REGION Network 50: End if not ready to next step
   // no SCL statement known for JumpNot: written as a call
   JumpNot(in := #POWER_STATE >= 90, label := END);
END_REGION

REGION Network 51: OPERATION
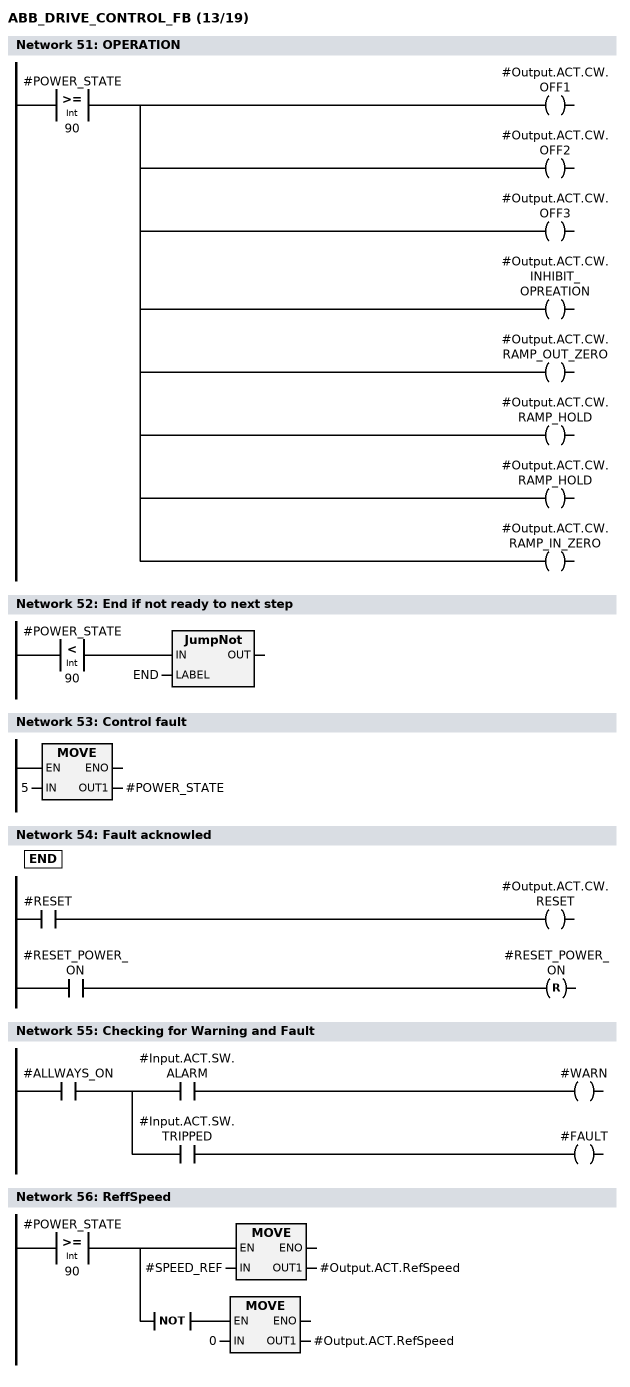
   RUNG wire#powerrail
      { S7_Templates := "SrcType := Int" } GE_Contact(in1 := #POWER_STATE, in2 := 90)
      wire#w1
      Coil( #Output.ACT.CW.OFF1 )
   END_RUNG
   RUNG wire#w1
      Coil( #Output.ACT.CW.OFF2 )
   END_RUNG
   RUNG wire#w1
      Coil( #Output.ACT.CW.OFF3 )
   END_RUNG
   RUNG wire#w1
      Coil( #Output.ACT.CW.INHIBIT_OPREATION )
   END_RUNG
   RUNG wire#w1
      Coil( #Output.ACT.CW.RAMP_OUT_ZERO )
   END_RUNG
   RUNG wire#w1
      Coil( #Output.ACT.CW.RAMP_HOLD )
   END_RUNG
   RUNG wire#w1
      Coil( #Output.ACT.CW.RAMP_HOLD )
   END_RUNG
   RUNG wire#w1
      Coil( #Output.ACT.CW.RAMP_IN_ZERO )
   END_RUNG
   // the same network as SCL:
   #Output.ACT.CW.OFF1 := #POWER_STATE >= 90;
   #Output.ACT.CW.OFF2 := #Output.ACT.CW.OFF1;
   #Output.ACT.CW.OFF3 := #Output.ACT.CW.OFF1;
   #Output.ACT.CW.INHIBIT_OPREATION := #Output.ACT.CW.OFF1;
   #Output.ACT.CW.RAMP_OUT_ZERO := #Output.ACT.CW.OFF1;
   #Output.ACT.CW.RAMP_HOLD := #Output.ACT.CW.OFF1;
   #Output.ACT.CW.RAMP_HOLD := #Output.ACT.CW.OFF1;
   #Output.ACT.CW.RAMP_IN_ZERO := #Output.ACT.CW.OFF1;
END_REGION

REGION Network 52: End if not ready to next step
   // no SCL statement known for JumpNot: written as a call
   JumpNot(in := #POWER_STATE < 90, label := END);
END_REGION

REGION Network 53: Control fault
   RUNG wire#powerrail
      { S7_GenerateENO := "TRUE" } Move(in := 5, out1 => #POWER_STATE)
   END_RUNG
   // the same network as SCL:
   #POWER_STATE := 5;
END_REGION

REGION Network 54: Fault acknowled
   Label( END )
   RUNG wire#powerrail
      Contact( #RESET )
      Coil( #Output.ACT.CW.RESET )
   END_RUNG
   RUNG wire#powerrail
      Contact( #RESET_POWER_ON )
      R_Coil( #RESET_POWER_ON )
   END_RUNG
   // the same network as SCL:
   END:
   #Output.ACT.CW.RESET := #RESET;
   IF #RESET_POWER_ON THEN #RESET_POWER_ON := FALSE; END_IF;
END_REGION

REGION Network 55: Checking for Warning and Fault
   RUNG wire#powerrail
      Contact( #ALLWAYS_ON )
      wire#w1
      Contact( #Input.ACT.SW.ALARM )
      Coil( #WARN )
   END_RUNG
   RUNG wire#w1
      Contact( #Input.ACT.SW.TRIPPED )
      Coil( #FAULT )
   END_RUNG
   // the same network as SCL:
   #WARN := #ALLWAYS_ON AND #Input.ACT.SW.ALARM;
   #FAULT := #ALLWAYS_ON AND #Input.ACT.SW.TRIPPED;
END_REGION

REGION Network 56: ReffSpeed
   RUNG wire#powerrail
      { S7_Templates := "SrcType := Int" } GE_Contact(in1 := #POWER_STATE, in2 := 90)
      wire#w1
      { S7_GenerateENO := "TRUE" } Move(in := #SPEED_REF, out1 => #Output.ACT.RefSpeed)
   END_RUNG
   RUNG wire#w1
      Not()
      { S7_GenerateENO := "TRUE" } Move(in := 0, out1 => #Output.ACT.RefSpeed)
   END_RUNG
   // the same network as SCL:
   #_w1 := #POWER_STATE >= 90;
   IF #_w1 THEN #Output.ACT.RefSpeed := #SPEED_REF; END_IF;
   IF NOT #_w1 THEN #Output.ACT.RefSpeed := 0; END_IF;
END_REGION

REGION Network 57: Write values PPO1 Fixed area
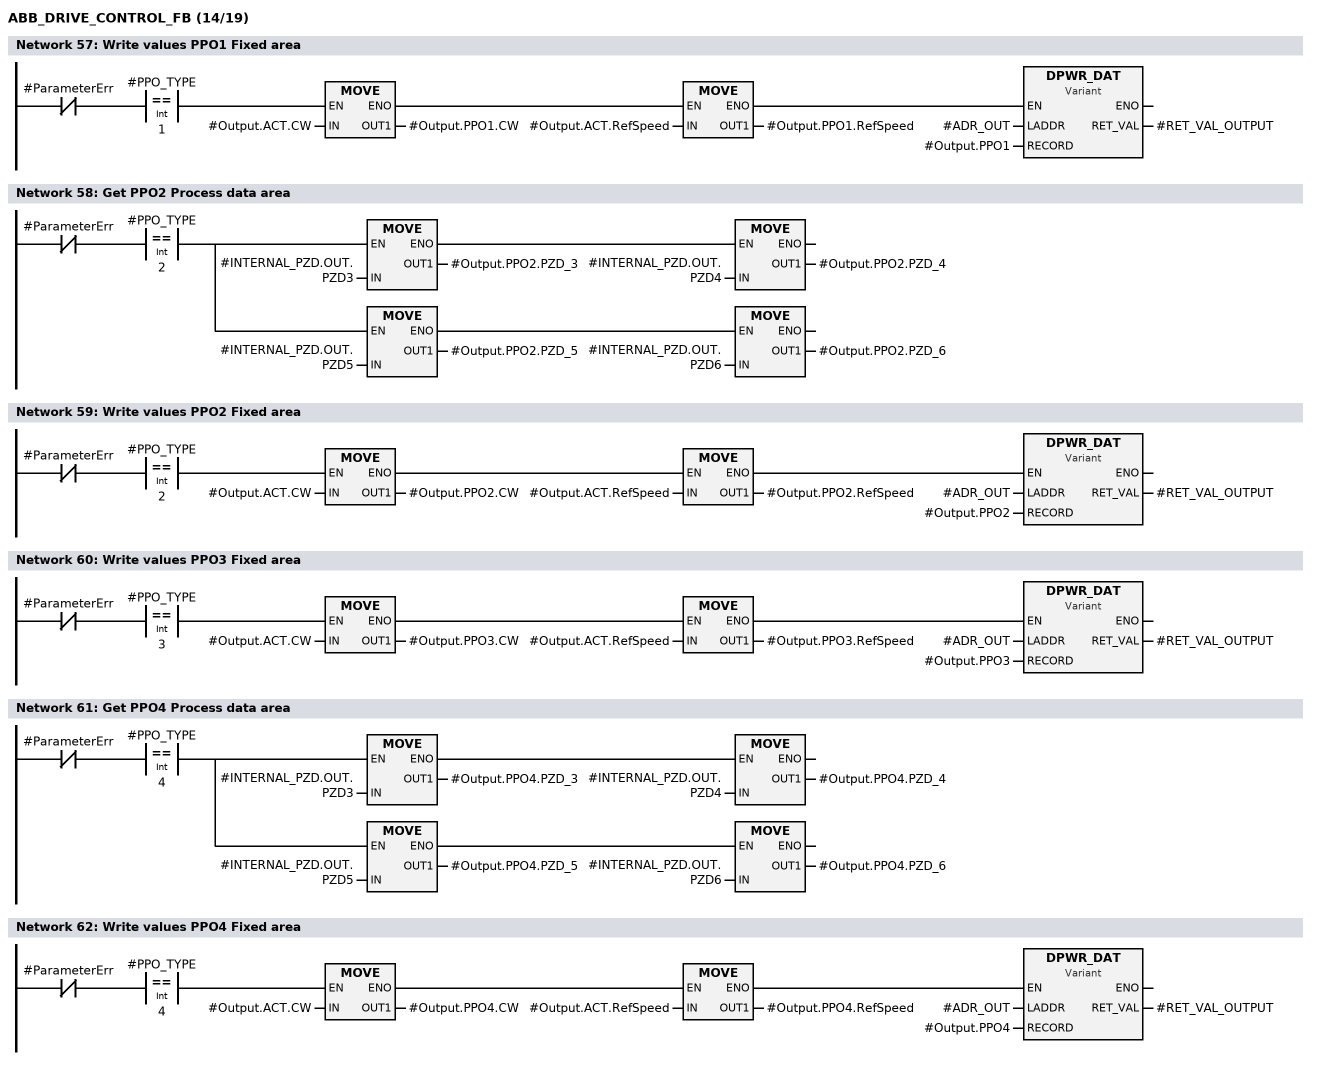
   RUNG wire#powerrail
      I_Contact( #ParameterErr )
      { S7_Templates := "SrcType := Int" } EQ_Contact(in1 := #PPO_TYPE, in2 := 1)
      { S7_GenerateENO := "TRUE" } Move(in := #Output.ACT.CW, out1 => #Output.PPO1.CW)
      { S7_GenerateENO := "TRUE" } Move(in := #Output.ACT.RefSpeed, out1 => #Output.PPO1.RefSpeed)
      { S7_Templates := "[ptr_type := Variant, laddr_type := HW_IO]" } DPWR_DAT(LADDR := #ADR_OUT, RECORD := #Output.PPO1, RET_VAL => #RET_VAL_OUTPUT)
   END_RUNG
   // the same network as SCL:
   // ENO of a box is taken as its EN; it also drops when the box reports an error
   IF NOT #ParameterErr AND (#PPO_TYPE = 1) THEN
       #Output.PPO1.CW := #Output.ACT.CW;
       #Output.PPO1.RefSpeed := #Output.ACT.RefSpeed;
       #RET_VAL_OUTPUT := DPWR_DAT(LADDR := #ADR_OUT, RECORD := #Output.PPO1);
   END_IF;
END_REGION

REGION Network 58: Get PPO2 Process data area
   RUNG wire#powerrail
      I_Contact( #ParameterErr )
      { S7_Templates := "SrcType := Int" } EQ_Contact(in1 := #PPO_TYPE, in2 := 2)
      wire#w1
      { S7_GenerateENO := "TRUE" } Move(in := #INTERNAL_PZD.OUT.PZD3, out1 => #Output.PPO2.PZD_3)
      { S7_GenerateENO := "TRUE" } Move(in := #INTERNAL_PZD.OUT.PZD4, out1 => #Output.PPO2.PZD_4)
   END_RUNG
   RUNG wire#w1
      { S7_GenerateENO := "TRUE" } Move(in := #INTERNAL_PZD.OUT.PZD5, out1 => #Output.PPO2.PZD_5)
      { S7_GenerateENO := "TRUE" } Move(in := #INTERNAL_PZD.OUT.PZD6, out1 => #Output.PPO2.PZD_6)
   END_RUNG
   // the same network as SCL:
   // ENO of a box is taken as its EN; it also drops when the box reports an error
   IF NOT #ParameterErr AND (#PPO_TYPE = 2) THEN
       #Output.PPO2.PZD_3 := #INTERNAL_PZD.OUT.PZD3;
       #Output.PPO2.PZD_4 := #INTERNAL_PZD.OUT.PZD4;
       #Output.PPO2.PZD_5 := #INTERNAL_PZD.OUT.PZD5;
       #Output.PPO2.PZD_6 := #INTERNAL_PZD.OUT.PZD6;
   END_IF;
END_REGION

REGION Network 59: Write values PPO2 Fixed area
   RUNG wire#powerrail
      I_Contact( #ParameterErr )
      { S7_Templates := "SrcType := Int" } EQ_Contact(in1 := #PPO_TYPE, in2 := 2)
      { S7_GenerateENO := "TRUE" } Move(in := #Output.ACT.CW, out1 => #Output.PPO2.CW)
      { S7_GenerateENO := "TRUE" } Move(in := #Output.ACT.RefSpeed, out1 => #Output.PPO2.RefSpeed)
      { S7_Templates := "[ptr_type := Variant, laddr_type := HW_IO]" } DPWR_DAT(LADDR := #ADR_OUT, RECORD := #Output.PPO2, RET_VAL => #RET_VAL_OUTPUT)
   END_RUNG
   // the same network as SCL:
   // ENO of a box is taken as its EN; it also drops when the box reports an error
   IF NOT #ParameterErr AND (#PPO_TYPE = 2) THEN
       #Output.PPO2.CW := #Output.ACT.CW;
       #Output.PPO2.RefSpeed := #Output.ACT.RefSpeed;
       #RET_VAL_OUTPUT := DPWR_DAT(LADDR := #ADR_OUT, RECORD := #Output.PPO2);
   END_IF;
END_REGION

REGION Network 60: Write values PPO3 Fixed area
   RUNG wire#powerrail
      I_Contact( #ParameterErr )
      { S7_Templates := "SrcType := Int" } EQ_Contact(in1 := #PPO_TYPE, in2 := 3)
      { S7_GenerateENO := "TRUE" } Move(in := #Output.ACT.CW, out1 => #Output.PPO3.CW)
      { S7_GenerateENO := "TRUE" } Move(in := #Output.ACT.RefSpeed, out1 => #Output.PPO3.RefSpeed)
      { S7_Templates := "[ptr_type := Variant, laddr_type := HW_IO]" } DPWR_DAT(LADDR := #ADR_OUT, RECORD := #Output.PPO3, RET_VAL => #RET_VAL_OUTPUT)
   END_RUNG
   // the same network as SCL:
   // ENO of a box is taken as its EN; it also drops when the box reports an error
   IF NOT #ParameterErr AND (#PPO_TYPE = 3) THEN
       #Output.PPO3.CW := #Output.ACT.CW;
       #Output.PPO3.RefSpeed := #Output.ACT.RefSpeed;
       #RET_VAL_OUTPUT := DPWR_DAT(LADDR := #ADR_OUT, RECORD := #Output.PPO3);
   END_IF;
END_REGION

REGION Network 61: Get PPO4 Process data area
   RUNG wire#powerrail
      I_Contact( #ParameterErr )
      { S7_Templates := "SrcType := Int" } EQ_Contact(in1 := #PPO_TYPE, in2 := 4)
      wire#w1
      { S7_GenerateENO := "TRUE" } Move(in := #INTERNAL_PZD.OUT.PZD3, out1 => #Output.PPO4.PZD_3)
      { S7_GenerateENO := "TRUE" } Move(in := #INTERNAL_PZD.OUT.PZD4, out1 => #Output.PPO4.PZD_4)
   END_RUNG
   RUNG wire#w1
      { S7_GenerateENO := "TRUE" } Move(in := #INTERNAL_PZD.OUT.PZD5, out1 => #Output.PPO4.PZD_5)
      { S7_GenerateENO := "TRUE" } Move(in := #INTERNAL_PZD.OUT.PZD6, out1 => #Output.PPO4.PZD_6)
   END_RUNG
   // the same network as SCL:
   // ENO of a box is taken as its EN; it also drops when the box reports an error
   IF NOT #ParameterErr AND (#PPO_TYPE = 4) THEN
       #Output.PPO4.PZD_3 := #INTERNAL_PZD.OUT.PZD3;
       #Output.PPO4.PZD_4 := #INTERNAL_PZD.OUT.PZD4;
       #Output.PPO4.PZD_5 := #INTERNAL_PZD.OUT.PZD5;
       #Output.PPO4.PZD_6 := #INTERNAL_PZD.OUT.PZD6;
   END_IF;
END_REGION

REGION Network 62: Write values PPO4 Fixed area
   RUNG wire#powerrail
      I_Contact( #ParameterErr )
      { S7_Templates := "SrcType := Int" } EQ_Contact(in1 := #PPO_TYPE, in2 := 4)
      { S7_GenerateENO := "TRUE" } Move(in := #Output.ACT.CW, out1 => #Output.PPO4.CW)
      { S7_GenerateENO := "TRUE" } Move(in := #Output.ACT.RefSpeed, out1 => #Output.PPO4.RefSpeed)
      { S7_Templates := "[ptr_type := Variant, laddr_type := HW_IO]" } DPWR_DAT(LADDR := #ADR_OUT, RECORD := #Output.PPO4, RET_VAL => #RET_VAL_OUTPUT)
   END_RUNG
   // the same network as SCL:
   // ENO of a box is taken as its EN; it also drops when the box reports an error
   IF NOT #ParameterErr AND (#PPO_TYPE = 4) THEN
       #Output.PPO4.CW := #Output.ACT.CW;
       #Output.PPO4.RefSpeed := #Output.ACT.RefSpeed;
       #RET_VAL_OUTPUT := DPWR_DAT(LADDR := #ADR_OUT, RECORD := #Output.PPO4);
   END_IF;
END_REGION

REGION Network 63: Get PPO5 Process data area
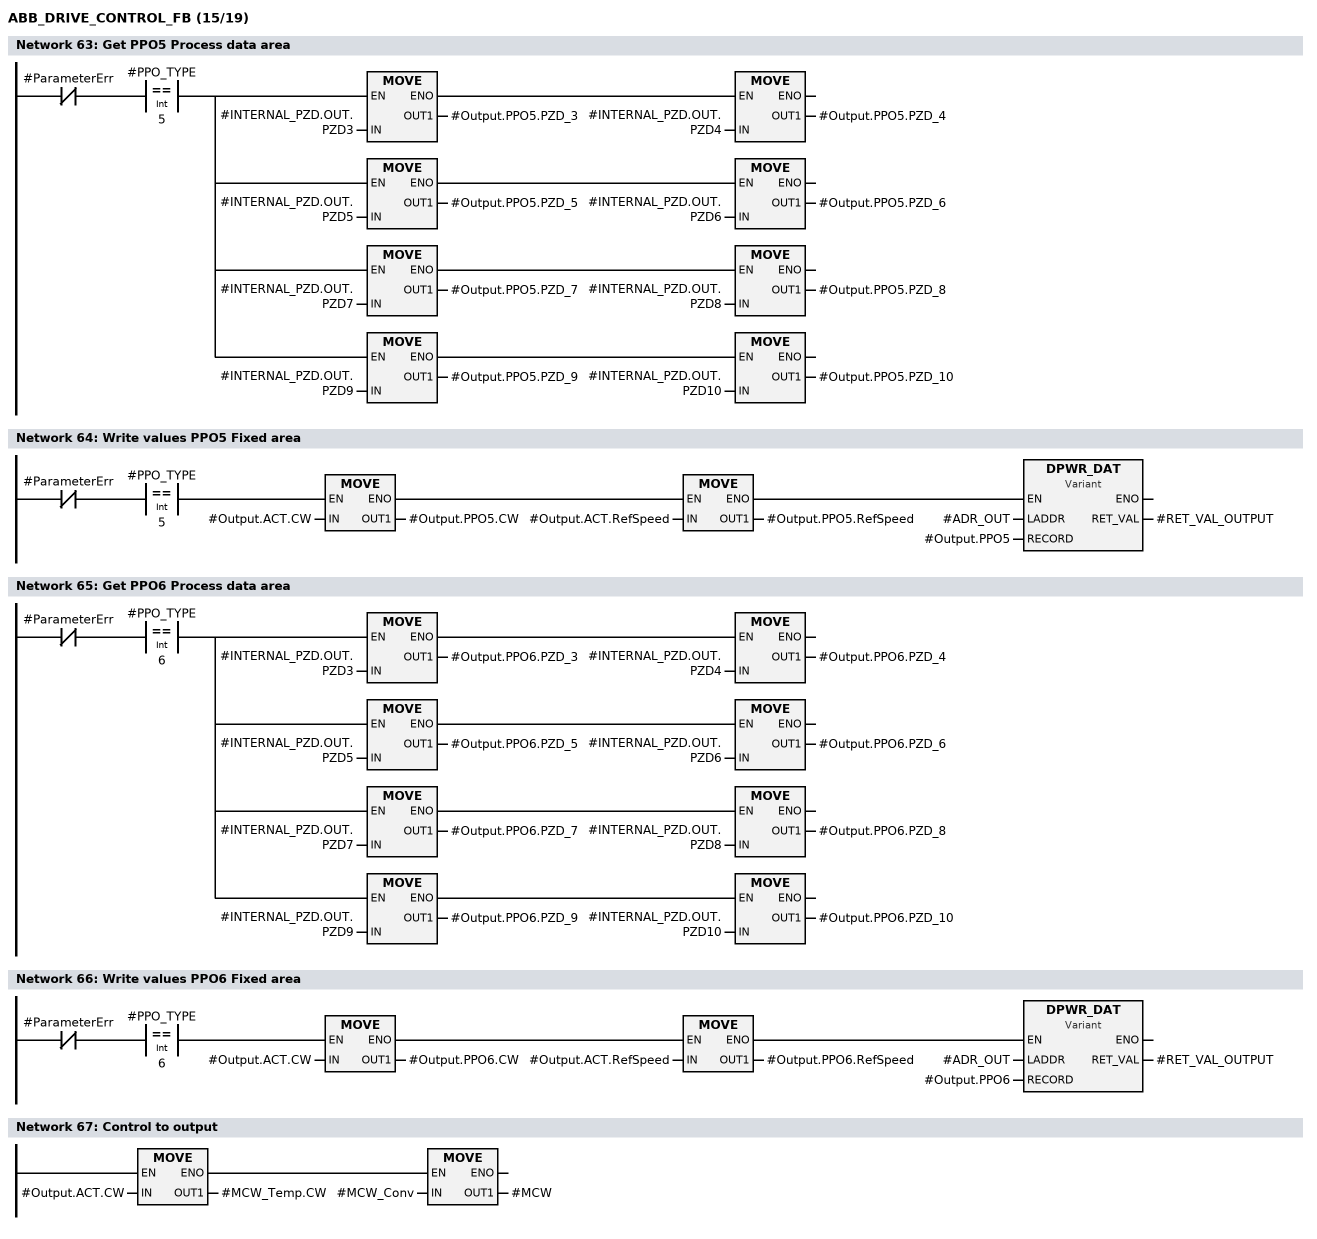
   RUNG wire#powerrail
      I_Contact( #ParameterErr )
      { S7_Templates := "SrcType := Int" } EQ_Contact(in1 := #PPO_TYPE, in2 := 5)
      wire#w1
      { S7_GenerateENO := "TRUE" } Move(in := #INTERNAL_PZD.OUT.PZD3, out1 => #Output.PPO5.PZD_3)
      { S7_GenerateENO := "TRUE" } Move(in := #INTERNAL_PZD.OUT.PZD4, out1 => #Output.PPO5.PZD_4)
   END_RUNG
   RUNG wire#w1
      { S7_GenerateENO := "TRUE" } Move(in := #INTERNAL_PZD.OUT.PZD5, out1 => #Output.PPO5.PZD_5)
      { S7_GenerateENO := "TRUE" } Move(in := #INTERNAL_PZD.OUT.PZD6, out1 => #Output.PPO5.PZD_6)
   END_RUNG
   RUNG wire#w1
      { S7_GenerateENO := "TRUE" } Move(in := #INTERNAL_PZD.OUT.PZD7, out1 => #Output.PPO5.PZD_7)
      { S7_GenerateENO := "TRUE" } Move(in := #INTERNAL_PZD.OUT.PZD8, out1 => #Output.PPO5.PZD_8)
   END_RUNG
   RUNG wire#w1
      { S7_GenerateENO := "TRUE" } Move(in := #INTERNAL_PZD.OUT.PZD9, out1 => #Output.PPO5.PZD_9)
      { S7_GenerateENO := "TRUE" } Move(in := #INTERNAL_PZD.OUT.PZD10, out1 => #Output.PPO5.PZD_10)
   END_RUNG
   // the same network as SCL:
   // ENO of a box is taken as its EN; it also drops when the box reports an error
   IF NOT #ParameterErr AND (#PPO_TYPE = 5) THEN
       #Output.PPO5.PZD_3 := #INTERNAL_PZD.OUT.PZD3;
       #Output.PPO5.PZD_4 := #INTERNAL_PZD.OUT.PZD4;
       #Output.PPO5.PZD_5 := #INTERNAL_PZD.OUT.PZD5;
       #Output.PPO5.PZD_6 := #INTERNAL_PZD.OUT.PZD6;
       #Output.PPO5.PZD_7 := #INTERNAL_PZD.OUT.PZD7;
       #Output.PPO5.PZD_8 := #INTERNAL_PZD.OUT.PZD8;
       #Output.PPO5.PZD_9 := #INTERNAL_PZD.OUT.PZD9;
       #Output.PPO5.PZD_10 := #INTERNAL_PZD.OUT.PZD10;
   END_IF;
END_REGION

REGION Network 64: Write values PPO5 Fixed area
   RUNG wire#powerrail
      I_Contact( #ParameterErr )
      { S7_Templates := "SrcType := Int" } EQ_Contact(in1 := #PPO_TYPE, in2 := 5)
      { S7_GenerateENO := "TRUE" } Move(in := #Output.ACT.CW, out1 => #Output.PPO5.CW)
      { S7_GenerateENO := "TRUE" } Move(in := #Output.ACT.RefSpeed, out1 => #Output.PPO5.RefSpeed)
      { S7_Templates := "[ptr_type := Variant, laddr_type := HW_IO]" } DPWR_DAT(LADDR := #ADR_OUT, RECORD := #Output.PPO5, RET_VAL => #RET_VAL_OUTPUT)
   END_RUNG
   // the same network as SCL:
   // ENO of a box is taken as its EN; it also drops when the box reports an error
   IF NOT #ParameterErr AND (#PPO_TYPE = 5) THEN
       #Output.PPO5.CW := #Output.ACT.CW;
       #Output.PPO5.RefSpeed := #Output.ACT.RefSpeed;
       #RET_VAL_OUTPUT := DPWR_DAT(LADDR := #ADR_OUT, RECORD := #Output.PPO5);
   END_IF;
END_REGION

REGION Network 65: Get PPO6 Process data area
   RUNG wire#powerrail
      I_Contact( #ParameterErr )
      { S7_Templates := "SrcType := Int" } EQ_Contact(in1 := #PPO_TYPE, in2 := 6)
      wire#w1
      { S7_GenerateENO := "TRUE" } Move(in := #INTERNAL_PZD.OUT.PZD3, out1 => #Output.PPO6.PZD_3)
      { S7_GenerateENO := "TRUE" } Move(in := #INTERNAL_PZD.OUT.PZD4, out1 => #Output.PPO6.PZD_4)
   END_RUNG
   RUNG wire#w1
      { S7_GenerateENO := "TRUE" } Move(in := #INTERNAL_PZD.OUT.PZD5, out1 => #Output.PPO6.PZD_5)
      { S7_GenerateENO := "TRUE" } Move(in := #INTERNAL_PZD.OUT.PZD6, out1 => #Output.PPO6.PZD_6)
   END_RUNG
   RUNG wire#w1
      { S7_GenerateENO := "TRUE" } Move(in := #INTERNAL_PZD.OUT.PZD7, out1 => #Output.PPO6.PZD_7)
      { S7_GenerateENO := "TRUE" } Move(in := #INTERNAL_PZD.OUT.PZD8, out1 => #Output.PPO6.PZD_8)
   END_RUNG
   RUNG wire#w1
      { S7_GenerateENO := "TRUE" } Move(in := #INTERNAL_PZD.OUT.PZD9, out1 => #Output.PPO6.PZD_9)
      { S7_GenerateENO := "TRUE" } Move(in := #INTERNAL_PZD.OUT.PZD10, out1 => #Output.PPO6.PZD_10)
   END_RUNG
   // the same network as SCL:
   // ENO of a box is taken as its EN; it also drops when the box reports an error
   IF NOT #ParameterErr AND (#PPO_TYPE = 6) THEN
       #Output.PPO6.PZD_3 := #INTERNAL_PZD.OUT.PZD3;
       #Output.PPO6.PZD_4 := #INTERNAL_PZD.OUT.PZD4;
       #Output.PPO6.PZD_5 := #INTERNAL_PZD.OUT.PZD5;
       #Output.PPO6.PZD_6 := #INTERNAL_PZD.OUT.PZD6;
       #Output.PPO6.PZD_7 := #INTERNAL_PZD.OUT.PZD7;
       #Output.PPO6.PZD_8 := #INTERNAL_PZD.OUT.PZD8;
       #Output.PPO6.PZD_9 := #INTERNAL_PZD.OUT.PZD9;
       #Output.PPO6.PZD_10 := #INTERNAL_PZD.OUT.PZD10;
   END_IF;
END_REGION

REGION Network 66: Write values PPO6 Fixed area
   RUNG wire#powerrail
      I_Contact( #ParameterErr )
      { S7_Templates := "SrcType := Int" } EQ_Contact(in1 := #PPO_TYPE, in2 := 6)
      { S7_GenerateENO := "TRUE" } Move(in := #Output.ACT.CW, out1 => #Output.PPO6.CW)
      { S7_GenerateENO := "TRUE" } Move(in := #Output.ACT.RefSpeed, out1 => #Output.PPO6.RefSpeed)
      { S7_Templates := "[ptr_type := Variant, laddr_type := HW_IO]" } DPWR_DAT(LADDR := #ADR_OUT, RECORD := #Output.PPO6, RET_VAL => #RET_VAL_OUTPUT)
   END_RUNG
   // the same network as SCL:
   // ENO of a box is taken as its EN; it also drops when the box reports an error
   IF NOT #ParameterErr AND (#PPO_TYPE = 6) THEN
       #Output.PPO6.CW := #Output.ACT.CW;
       #Output.PPO6.RefSpeed := #Output.ACT.RefSpeed;
       #RET_VAL_OUTPUT := DPWR_DAT(LADDR := #ADR_OUT, RECORD := #Output.PPO6);
   END_IF;
END_REGION

REGION Network 67: Control to output
   RUNG wire#powerrail
      { S7_GenerateENO := "TRUE" } Move(in := #Output.ACT.CW, out1 => #MCW_Temp.CW)
      { S7_GenerateENO := "TRUE" } Move(in := #MCW_Conv, out1 => #MCW)
   END_RUNG
   // the same network as SCL:
   // ENO of a box is taken as its EN; it also drops when the box reports an error
   #MCW_Temp.CW := #Output.ACT.CW;
   #MCW := #MCW_Conv;
END_REGION

REGION Network 68: Write parameters area DP-V0
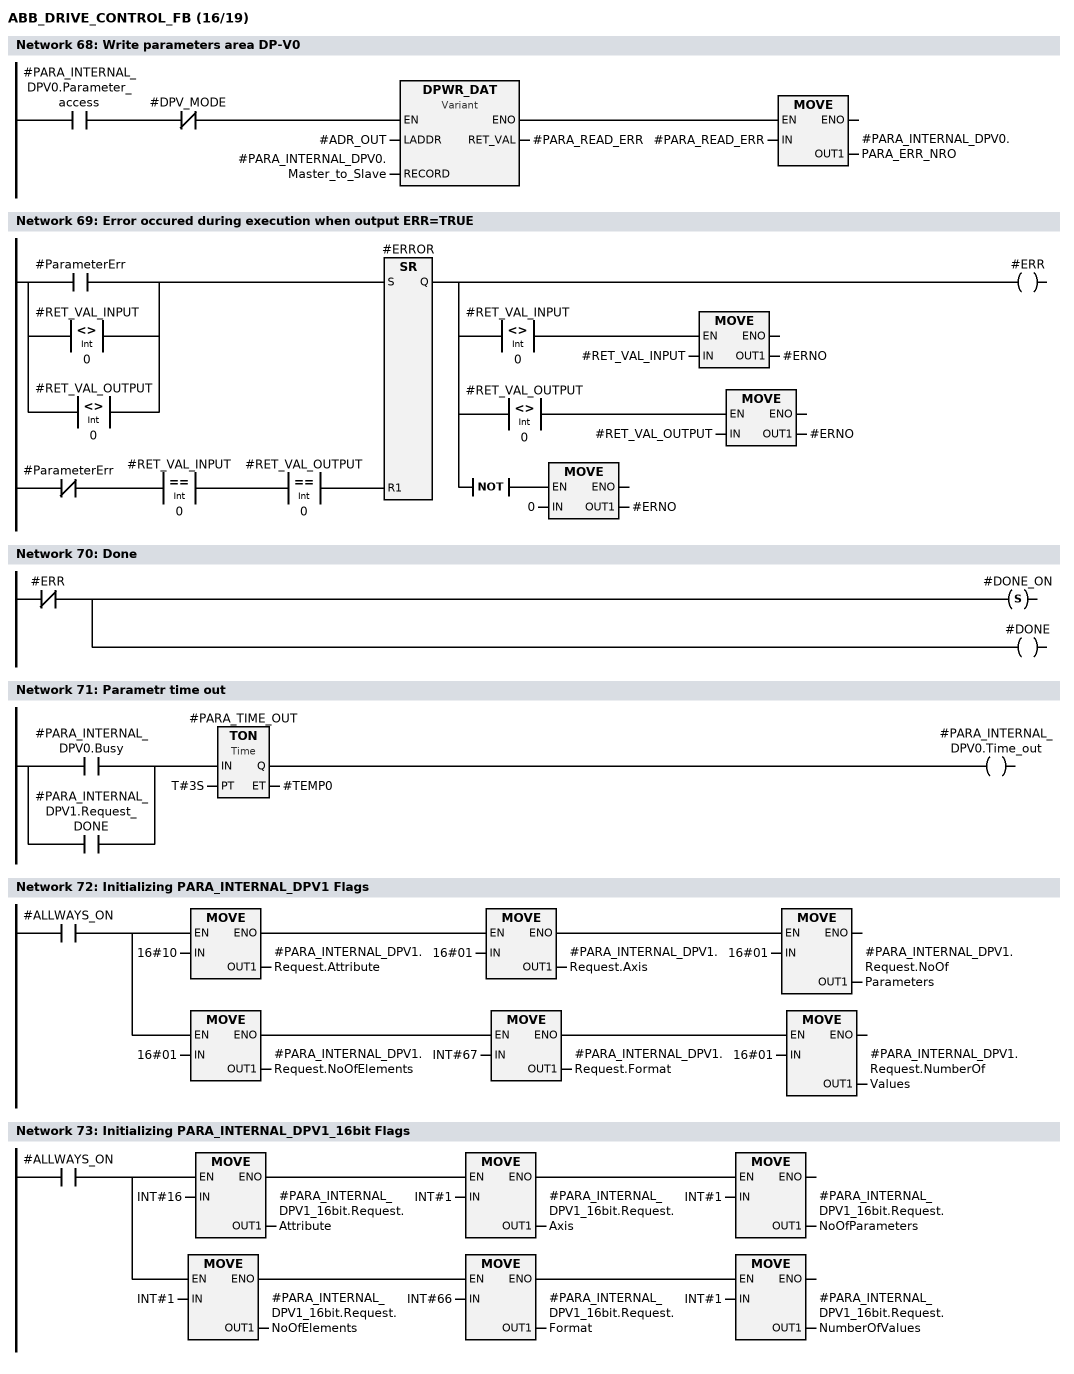
   RUNG wire#powerrail
      Contact( #PARA_INTERNAL_DPV0.Parameter_access )
      I_Contact( #DPV_MODE )
      { S7_Templates := "[ptr_type := Variant, laddr_type := HW_IO]" } DPWR_DAT(LADDR := #ADR_OUT, RECORD := #PARA_INTERNAL_DPV0.Master_to_Slave, RET_VAL => #PARA_READ_ERR)
      { S7_GenerateENO := "TRUE" } Move(in := #PARA_READ_ERR, out1 => #PARA_INTERNAL_DPV0.PARA_ERR_NRO)
   END_RUNG
   // the same network as SCL:
   #PARA_READ_ERR := DPWR_DAT(EN := #PARA_INTERNAL_DPV0.Parameter_access AND NOT #DPV_MODE,
                           LADDR := #ADR_OUT,
                           RECORD := #PARA_INTERNAL_DPV0.Master_to_Slave,
                           ENO => #_w1);
   IF #_w1 THEN #PARA_INTERNAL_DPV0.PARA_ERR_NRO := #PARA_READ_ERR; END_IF;
END_REGION

REGION Network 69: Error occured during execution when output ERR=TRUE
   RUNG wire#powerrail
      Contact( #ParameterErr )
      wire#w1
      S_SR(operand := #ERROR, r1 := wire#w2)
      wire#w3
      Coil( #ERR )
   END_RUNG
   RUNG wire#powerrail
      { S7_Templates := "SrcType := Int" } NE_Contact(in1 := #RET_VAL_INPUT, in2 := 0)
   END_RUNG wire#w1
   RUNG wire#powerrail
      { S7_Templates := "SrcType := Int" } NE_Contact(in1 := #RET_VAL_OUTPUT, in2 := 0)
   END_RUNG wire#w1
   RUNG wire#powerrail
      I_Contact( #ParameterErr )
      { S7_Templates := "SrcType := Int" } EQ_Contact(in1 := #RET_VAL_INPUT, in2 := 0)
      { S7_Templates := "SrcType := Int" } EQ_Contact(in1 := #RET_VAL_OUTPUT, in2 := 0)
   END_RUNG wire#w2
   RUNG wire#w3
      { S7_Templates := "SrcType := Int" } NE_Contact(in1 := #RET_VAL_INPUT, in2 := 0)
      { S7_GenerateENO := "TRUE" } Move(in := #RET_VAL_INPUT, out1 => #ERNO)
   END_RUNG
   RUNG wire#w3
      { S7_Templates := "SrcType := Int" } NE_Contact(in1 := #RET_VAL_OUTPUT, in2 := 0)
      { S7_GenerateENO := "TRUE" } Move(in := #RET_VAL_OUTPUT, out1 => #ERNO)
   END_RUNG
   RUNG wire#w3
      Not()
      { S7_GenerateENO := "TRUE" } Move(in := 0, out1 => #ERNO)
   END_RUNG
   // the same network as SCL:
   IF #ParameterErr OR (#RET_VAL_INPUT <> 0) OR (#RET_VAL_OUTPUT <> 0) THEN
       #ERROR := TRUE;   // SR flip-flop
   END_IF;
   IF NOT #ParameterErr AND (#RET_VAL_INPUT = 0) AND (#RET_VAL_OUTPUT = 0) THEN #ERROR := FALSE; END_IF;
   #ERR := #ERROR;
   IF #ERROR AND (#RET_VAL_INPUT <> 0) THEN #ERNO := #RET_VAL_INPUT; END_IF;
   IF #ERROR AND (#RET_VAL_OUTPUT <> 0) THEN #ERNO := #RET_VAL_OUTPUT; END_IF;
   IF NOT #ERROR THEN #ERNO := 0; END_IF;
END_REGION

REGION Network 70: Done
   RUNG wire#powerrail
      I_Contact( #ERR )
      wire#w1
      S_Coil( #DONE_ON )
   END_RUNG
   RUNG wire#w1
      Coil( #DONE )
   END_RUNG
   // the same network as SCL:
   IF NOT #ERR THEN #DONE_ON := TRUE; END_IF;
   #DONE := NOT #ERR;
END_REGION

REGION Network 71: Parametr time out
   RUNG wire#powerrail
      Contact( #PARA_INTERNAL_DPV0.Busy )
      wire#w1
      { S7_Templates := "time_type := Time" } #PARA_TIME_OUT.TON(pt := T#3S, et => #TEMP0)
      Coil( #PARA_INTERNAL_DPV0.Time_out )
   END_RUNG
   RUNG wire#powerrail
      Contact( #PARA_INTERNAL_DPV1.Request_DONE )
   END_RUNG wire#w1
   // the same network as SCL:
   #PARA_TIME_OUT(IN := #PARA_INTERNAL_DPV0.Busy OR #PARA_INTERNAL_DPV1.Request_DONE, PT := T#3S, ET => #TEMP0);   // TON
   #PARA_INTERNAL_DPV0.Time_out := #PARA_TIME_OUT.Q;
END_REGION

REGION Network 72: Initializing PARA_INTERNAL_DPV1 Flags
   RUNG wire#powerrail
      Contact( #ALLWAYS_ON )
      wire#w1
      { S7_GenerateENO := "TRUE" } Move(in := 16#10, out1 => #PARA_INTERNAL_DPV1.Request.Attribute)
      { S7_GenerateENO := "TRUE" } Move(in := 16#01, out1 => #PARA_INTERNAL_DPV1.Request.Axis)
      { S7_GenerateENO := "TRUE" } Move(in := 16#01, out1 => #PARA_INTERNAL_DPV1.Request.NoOfParameters)
   END_RUNG
   RUNG wire#w1
      { S7_GenerateENO := "TRUE" } Move(in := 16#01, out1 => #PARA_INTERNAL_DPV1.Request.NoOfElements)
      { S7_GenerateENO := "TRUE" } Move(in := INT#67, out1 => #PARA_INTERNAL_DPV1.Request.Format)
      { S7_GenerateENO := "TRUE" } Move(in := 16#01, out1 => #PARA_INTERNAL_DPV1.Request.NumberOfValues)
   END_RUNG
   // the same network as SCL:
   // ENO of a box is taken as its EN; it also drops when the box reports an error
   IF #ALLWAYS_ON THEN
       #PARA_INTERNAL_DPV1.Request.Attribute := 16#10;
       #PARA_INTERNAL_DPV1.Request.Axis := 16#01;
       #PARA_INTERNAL_DPV1.Request.NoOfParameters := 16#01;
       #PARA_INTERNAL_DPV1.Request.NoOfElements := 16#01;
       #PARA_INTERNAL_DPV1.Request.Format := INT#67;
       #PARA_INTERNAL_DPV1.Request.NumberOfValues := 16#01;
   END_IF;
END_REGION

REGION Network 73: Initializing PARA_INTERNAL_DPV1_16bit Flags
   RUNG wire#powerrail
      Contact( #ALLWAYS_ON )
      wire#w1
      { S7_GenerateENO := "TRUE" } Move(in := INT#16, out1 => #PARA_INTERNAL_DPV1_16bit.Request.Attribute)
      { S7_GenerateENO := "TRUE" } Move(in := INT#1, out1 => #PARA_INTERNAL_DPV1_16bit.Request.Axis)
      { S7_GenerateENO := "TRUE" } Move(in := INT#1, out1 => #PARA_INTERNAL_DPV1_16bit.Request.NoOfParameters)
   END_RUNG
   RUNG wire#w1
      { S7_GenerateENO := "TRUE" } Move(in := INT#1, out1 => #PARA_INTERNAL_DPV1_16bit.Request.NoOfElements)
      { S7_GenerateENO := "TRUE" } Move(in := INT#66, out1 => #PARA_INTERNAL_DPV1_16bit.Request.Format)
      { S7_GenerateENO := "TRUE" } Move(in := INT#1, out1 => #PARA_INTERNAL_DPV1_16bit.Request.NumberOfValues)
   END_RUNG
   // the same network as SCL:
   // ENO of a box is taken as its EN; it also drops when the box reports an error
   IF #ALLWAYS_ON THEN
       #PARA_INTERNAL_DPV1_16bit.Request.Attribute := INT#16;
       #PARA_INTERNAL_DPV1_16bit.Request.Axis := INT#1;
       #PARA_INTERNAL_DPV1_16bit.Request.NoOfParameters := INT#1;
       #PARA_INTERNAL_DPV1_16bit.Request.NoOfElements := INT#1;
       #PARA_INTERNAL_DPV1_16bit.Request.Format := INT#66;
       #PARA_INTERNAL_DPV1_16bit.Request.NumberOfValues := INT#1;
   END_IF;
END_REGION

REGION Network 74: Read/Write request reference
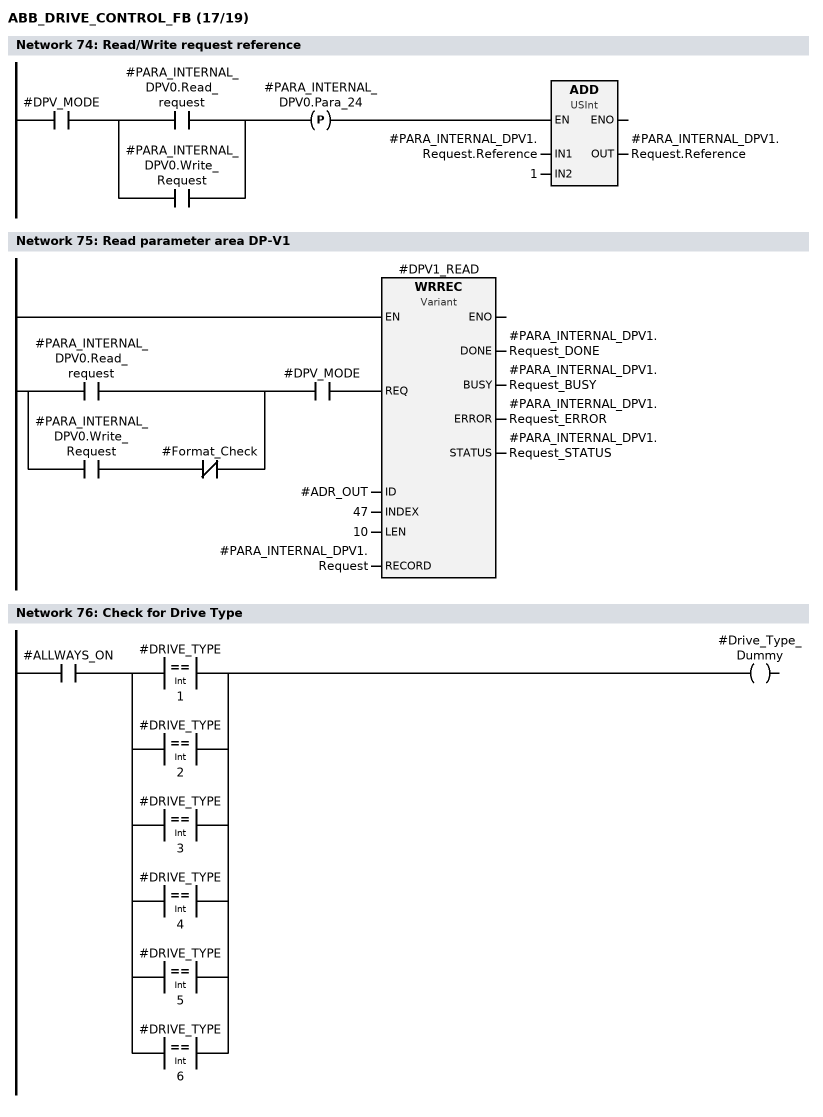
   RUNG wire#powerrail
      Contact( #DPV_MODE )
      wire#w1
      Contact( #PARA_INTERNAL_DPV0.Read_request )
      wire#w2
      P_Trig( #PARA_INTERNAL_DPV0.Para_24 )
      { S7_Templates := "SrcType := USInt"; S7_GenerateENO := "TRUE" } Add(in1 := #PARA_INTERNAL_DPV1.Request.Reference, in2 := 1, out => #PARA_INTERNAL_DPV1.Request.Reference)
   END_RUNG
   RUNG wire#w1
      Contact( #PARA_INTERNAL_DPV0.Write_Request )
   END_RUNG wire#w2
   // the same network as SCL:
   #_w1 := #DPV_MODE AND (#PARA_INTERNAL_DPV0.Read_request OR #PARA_INTERNAL_DPV0.Write_Request);
   #_w2 := #_w1 AND NOT #PARA_INTERNAL_DPV0.Para_24;   // rising edge
   #PARA_INTERNAL_DPV0.Para_24 := #_w1;
   IF #_w2 THEN #PARA_INTERNAL_DPV1.Request.Reference := #PARA_INTERNAL_DPV1.Request.Reference + 1; END_IF;
END_REGION

REGION Network 75: Read parameter area DP-V1
   RUNG wire#powerrail
      { S7_Templates := "[ptr_type := Variant, id_type := HW_IO, index_type := DInt, len_type := UInt]" } #DPV1_READ.WRREC(REQ := wire#w2, ID := #ADR_OUT, INDEX := 47, LEN := 10, RECORD := #PARA_INTERNAL_DPV1.Request, DONE => #PARA_INTERNAL_DPV1.Request_DONE, BUSY => #PARA_INTERNAL_DPV1.Request_BUSY, ERROR => #PARA_INTERNAL_DPV1.Request_ERROR, STATUS => #PARA_INTERNAL_DPV1.Request_STATUS)
   END_RUNG
   RUNG wire#powerrail
      Contact( #PARA_INTERNAL_DPV0.Read_request )
      wire#w1
      Contact( #DPV_MODE )
   END_RUNG wire#w2
   RUNG wire#powerrail
      Contact( #PARA_INTERNAL_DPV0.Write_Request )
      I_Contact( #Format_Check )
   END_RUNG wire#w1
   // the same network as SCL:
   #DPV1_READ(REQ := (#PARA_INTERNAL_DPV0.Read_request OR (#PARA_INTERNAL_DPV0.Write_Request AND NOT #Format_Check)) AND #DPV_MODE,   // WRREC
              ID := #ADR_OUT,
              INDEX := 47,
              LEN := 10,
              RECORD := #PARA_INTERNAL_DPV1.Request,
              DONE => #PARA_INTERNAL_DPV1.Request_DONE,
              BUSY => #PARA_INTERNAL_DPV1.Request_BUSY,
              ERROR => #PARA_INTERNAL_DPV1.Request_ERROR,
              STATUS => #PARA_INTERNAL_DPV1.Request_STATUS);
END_REGION

REGION Network 76: Check for Drive Type
   RUNG wire#powerrail
      Contact( #ALLWAYS_ON )
      wire#w1
      { S7_Templates := "SrcType := Int" } EQ_Contact(in1 := #DRIVE_TYPE, in2 := 1)
      wire#w2
      Coil( #Drive_Type_Dummy )
   END_RUNG
   RUNG wire#w1
      { S7_Templates := "SrcType := Int" } EQ_Contact(in1 := #DRIVE_TYPE, in2 := 2)
   END_RUNG wire#w2
   RUNG wire#w1
      { S7_Templates := "SrcType := Int" } EQ_Contact(in1 := #DRIVE_TYPE, in2 := 3)
   END_RUNG wire#w2
   RUNG wire#w1
      { S7_Templates := "SrcType := Int" } EQ_Contact(in1 := #DRIVE_TYPE, in2 := 4)
   END_RUNG wire#w2
   RUNG wire#w1
      { S7_Templates := "SrcType := Int" } EQ_Contact(in1 := #DRIVE_TYPE, in2 := 5)
   END_RUNG wire#w2
   RUNG wire#w1
      { S7_Templates := "SrcType := Int" } EQ_Contact(in1 := #DRIVE_TYPE, in2 := 6)
   END_RUNG wire#w2
   // the same network as SCL:
   #Drive_Type_Dummy := #ALLWAYS_ON AND ((#DRIVE_TYPE = 1) OR (#DRIVE_TYPE = 2) OR (#DRIVE_TYPE = 3) OR (#DRIVE_TYPE = 4) OR (#DRIVE_TYPE = 5) OR (#DRIVE_TYPE = 6));
END_REGION

REGION Network 77: Check for Drive Type
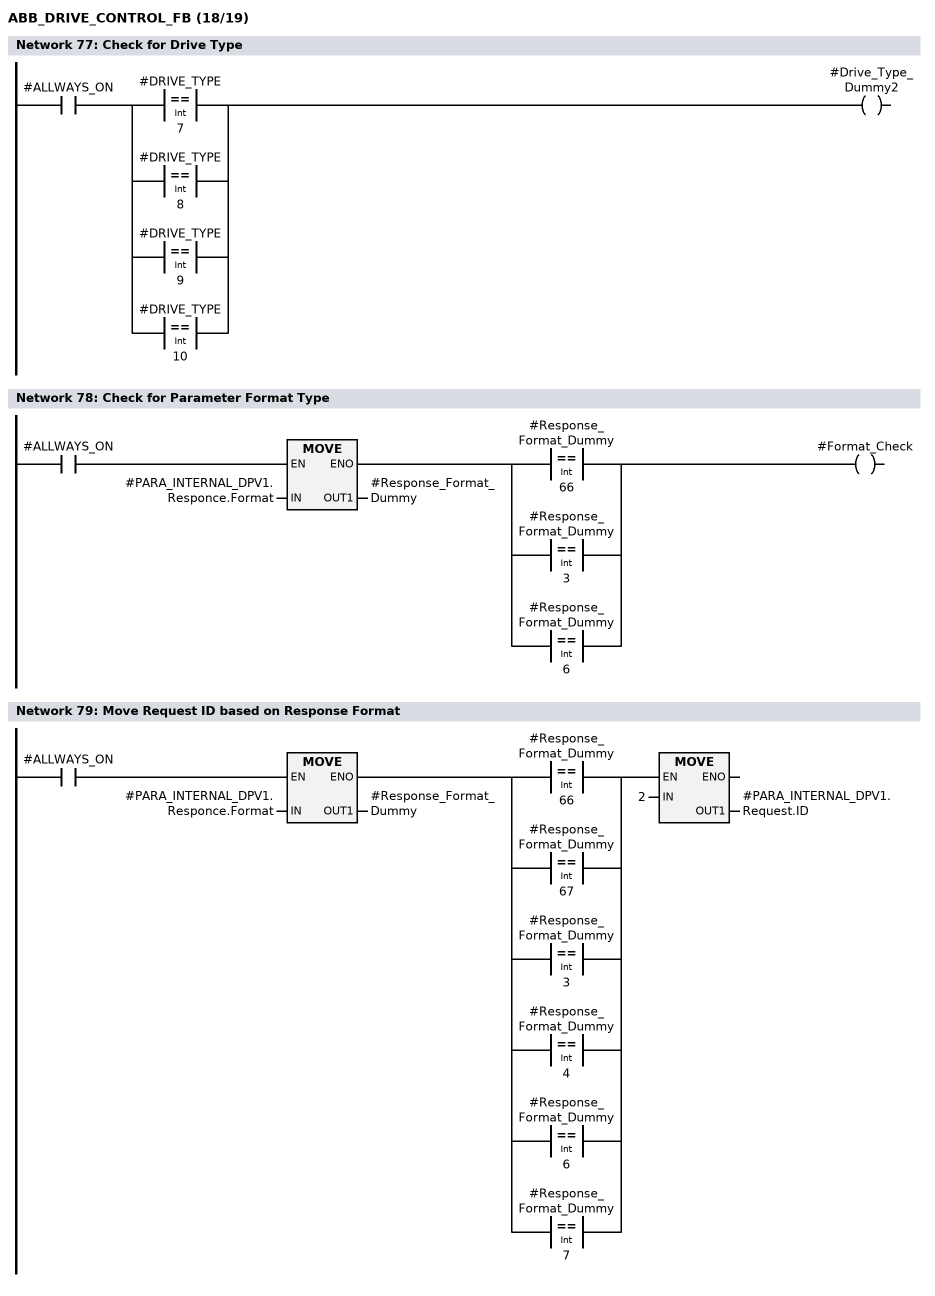
   RUNG wire#powerrail
      Contact( #ALLWAYS_ON )
      wire#w1
      { S7_Templates := "SrcType := Int" } EQ_Contact(in1 := #DRIVE_TYPE, in2 := 7)
      wire#w2
      Coil( #Drive_Type_Dummy2 )
   END_RUNG
   RUNG wire#w1
      { S7_Templates := "SrcType := Int" } EQ_Contact(in1 := #DRIVE_TYPE, in2 := 8)
   END_RUNG wire#w2
   RUNG wire#w1
      { S7_Templates := "SrcType := Int" } EQ_Contact(in1 := #DRIVE_TYPE, in2 := 9)
   END_RUNG wire#w2
   RUNG wire#w1
      { S7_Templates := "SrcType := Int" } EQ_Contact(in1 := #DRIVE_TYPE, in2 := 10)
   END_RUNG wire#w2
   // the same network as SCL:
   #Drive_Type_Dummy2 := #ALLWAYS_ON AND ((#DRIVE_TYPE = 7) OR (#DRIVE_TYPE = 8) OR (#DRIVE_TYPE = 9) OR (#DRIVE_TYPE = 10));
END_REGION

REGION Network 78: Check for Parameter Format Type
   RUNG wire#powerrail
      Contact( #ALLWAYS_ON )
      { S7_GenerateENO := "TRUE" } Move(in := #PARA_INTERNAL_DPV1.Responce.Format, out1 => #Response_Format_Dummy)
      wire#w1
      { S7_Templates := "SrcType := Int" } EQ_Contact(in1 := #Response_Format_Dummy, in2 := 66)
      wire#w2
      Coil( #Format_Check )
   END_RUNG
   RUNG wire#w1
      { S7_Templates := "SrcType := Int" } EQ_Contact(in1 := #Response_Format_Dummy, in2 := 3)
   END_RUNG wire#w2
   RUNG wire#w1
      { S7_Templates := "SrcType := Int" } EQ_Contact(in1 := #Response_Format_Dummy, in2 := 6)
   END_RUNG wire#w2
   // the same network as SCL:
   // ENO of a box is taken as its EN; it also drops when the box reports an error
   IF #ALLWAYS_ON THEN #Response_Format_Dummy := #PARA_INTERNAL_DPV1.Responce.Format; END_IF;
   #Format_Check := #ALLWAYS_ON AND ((#Response_Format_Dummy = 66) OR (#Response_Format_Dummy = 3) OR (#Response_Format_Dummy = 6));
END_REGION

REGION Network 79: Move Request ID based on Response Format
   RUNG wire#powerrail
      Contact( #ALLWAYS_ON )
      { S7_GenerateENO := "TRUE" } Move(in := #PARA_INTERNAL_DPV1.Responce.Format, out1 => #Response_Format_Dummy)
      wire#w1
      { S7_Templates := "SrcType := Int" } EQ_Contact(in1 := #Response_Format_Dummy, in2 := 66)
      wire#w2
      { S7_GenerateENO := "TRUE" } Move(in := 2, out1 => #PARA_INTERNAL_DPV1.Request.ID)
   END_RUNG
   RUNG wire#w1
      { S7_Templates := "SrcType := Int" } EQ_Contact(in1 := #Response_Format_Dummy, in2 := 67)
   END_RUNG wire#w2
   RUNG wire#w1
      { S7_Templates := "SrcType := Int" } EQ_Contact(in1 := #Response_Format_Dummy, in2 := 3)
   END_RUNG wire#w2
   RUNG wire#w1
      { S7_Templates := "SrcType := Int" } EQ_Contact(in1 := #Response_Format_Dummy, in2 := 4)
   END_RUNG wire#w2
   RUNG wire#w1
      { S7_Templates := "SrcType := Int" } EQ_Contact(in1 := #Response_Format_Dummy, in2 := 6)
   END_RUNG wire#w2
   RUNG wire#w1
      { S7_Templates := "SrcType := Int" } EQ_Contact(in1 := #Response_Format_Dummy, in2 := 7)
   END_RUNG wire#w2
   // the same network as SCL:
   // ENO of a box is taken as its EN; it also drops when the box reports an error
   IF #ALLWAYS_ON THEN #Response_Format_Dummy := #PARA_INTERNAL_DPV1.Responce.Format; END_IF;
   IF #ALLWAYS_ON AND ((#Response_Format_Dummy = 66) OR (#Response_Format_Dummy = 67) OR (#Response_Format_Dummy = 3) OR (#Response_Format_Dummy = 4) OR (#Response_Format_Dummy = 6) OR (#Response_Format_Dummy = 7)) THEN
       #PARA_INTERNAL_DPV1.Request.ID := 2;
   END_IF;
END_REGION

REGION Network 80: Check for Parameter Format Type
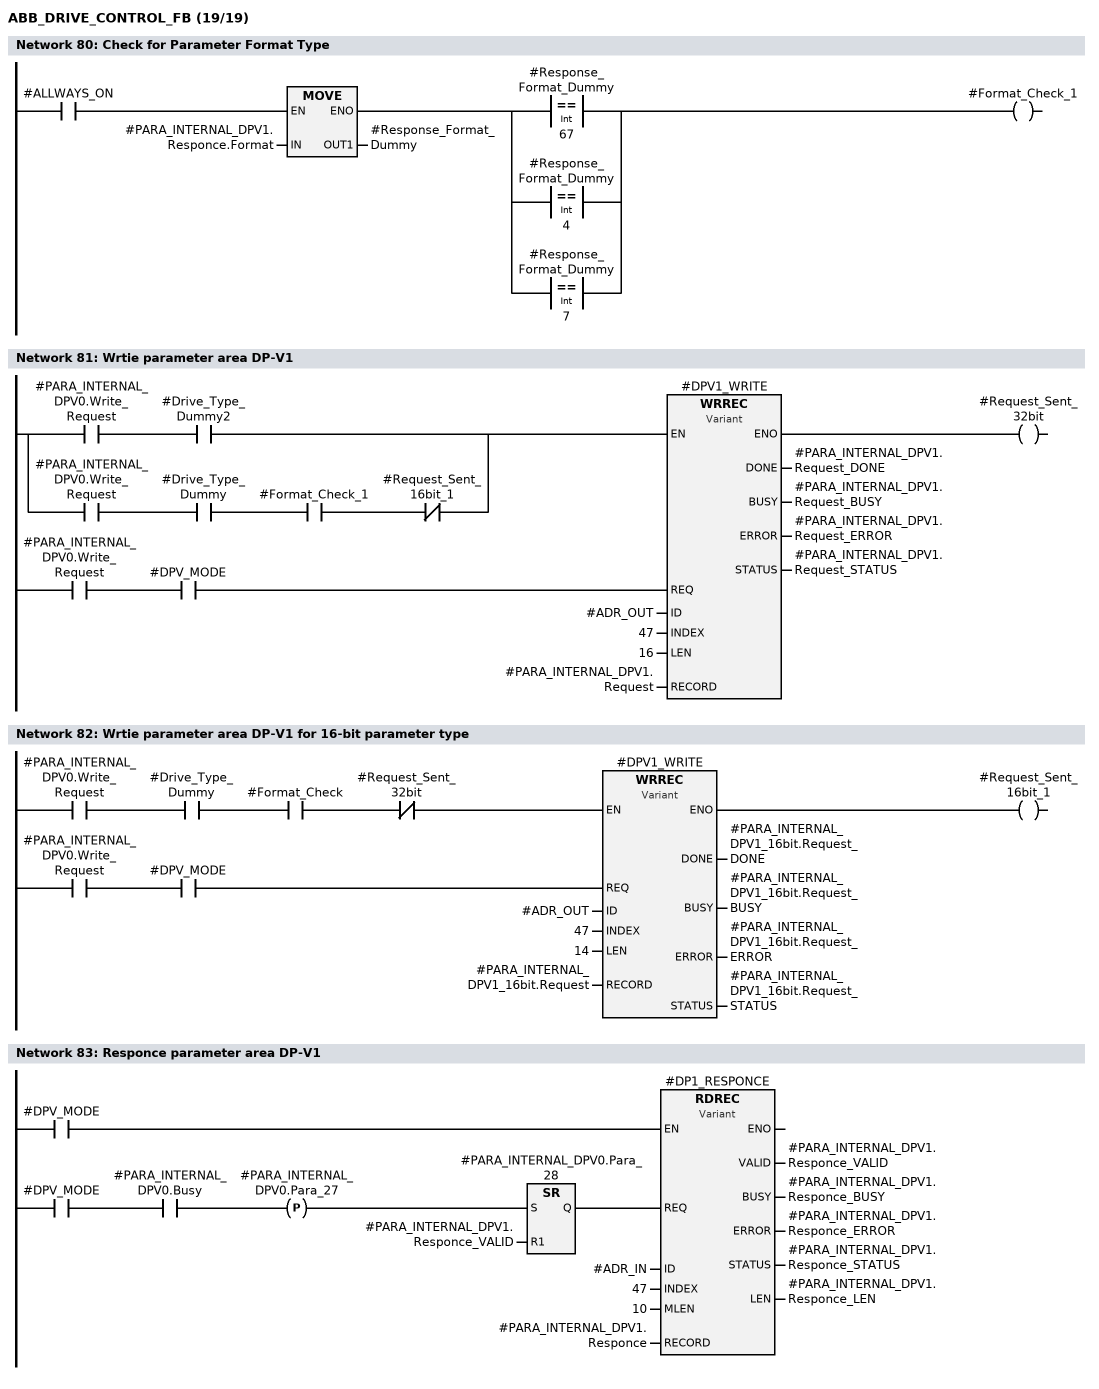
   RUNG wire#powerrail
      Contact( #ALLWAYS_ON )
      { S7_GenerateENO := "TRUE" } Move(in := #PARA_INTERNAL_DPV1.Responce.Format, out1 => #Response_Format_Dummy)
      wire#w1
      { S7_Templates := "SrcType := Int" } EQ_Contact(in1 := #Response_Format_Dummy, in2 := 67)
      wire#w2
      Coil( #Format_Check_1 )
   END_RUNG
   RUNG wire#w1
      { S7_Templates := "SrcType := Int" } EQ_Contact(in1 := #Response_Format_Dummy, in2 := 4)
   END_RUNG wire#w2
   RUNG wire#w1
      { S7_Templates := "SrcType := Int" } EQ_Contact(in1 := #Response_Format_Dummy, in2 := 7)
   END_RUNG wire#w2
   // the same network as SCL:
   // ENO of a box is taken as its EN; it also drops when the box reports an error
   IF #ALLWAYS_ON THEN #Response_Format_Dummy := #PARA_INTERNAL_DPV1.Responce.Format; END_IF;
   #Format_Check_1 := #ALLWAYS_ON AND ((#Response_Format_Dummy = 67) OR (#Response_Format_Dummy = 4) OR (#Response_Format_Dummy = 7));
END_REGION

REGION Network 81: Wrtie parameter area DP-V1
   RUNG wire#powerrail
      Contact( #PARA_INTERNAL_DPV0.Write_Request )
      Contact( #Drive_Type_Dummy2 )
      wire#w1
      { S7_Templates := "[ptr_type := Variant, id_type := HW_IO, index_type := DInt, len_type := UInt]" } #DPV1_WRITE.WRREC(REQ := wire#w2, ID := #ADR_OUT, INDEX := 47, LEN := 16, RECORD := #PARA_INTERNAL_DPV1.Request, DONE => #PARA_INTERNAL_DPV1.Request_DONE, BUSY => #PARA_INTERNAL_DPV1.Request_BUSY, ERROR => #PARA_INTERNAL_DPV1.Request_ERROR, STATUS => #PARA_INTERNAL_DPV1.Request_STATUS)
      Coil( #Request_Sent_32bit )
   END_RUNG
   RUNG wire#powerrail
      Contact( #PARA_INTERNAL_DPV0.Write_Request )
      Contact( #Drive_Type_Dummy )
      Contact( #Format_Check_1 )
      I_Contact( #Request_Sent_16bit_1 )
   END_RUNG wire#w1
   RUNG wire#powerrail
      Contact( #PARA_INTERNAL_DPV0.Write_Request )
      Contact( #DPV_MODE )
   END_RUNG wire#w2
   // the same network as SCL:
   #_w1 := (#PARA_INTERNAL_DPV0.Write_Request AND #Drive_Type_Dummy2) OR (#PARA_INTERNAL_DPV0.Write_Request AND #Drive_Type_Dummy AND #Format_Check_1 AND NOT #Request_Sent_16bit_1);
   #DPV1_WRITE(EN := #_w1,   // WRREC
               REQ := #PARA_INTERNAL_DPV0.Write_Request AND #DPV_MODE,
               ID := #ADR_OUT,
               INDEX := 47,
               LEN := 16,
               RECORD := #PARA_INTERNAL_DPV1.Request,
               DONE => #PARA_INTERNAL_DPV1.Request_DONE,
               BUSY => #PARA_INTERNAL_DPV1.Request_BUSY,
               ERROR => #PARA_INTERNAL_DPV1.Request_ERROR,
               STATUS => #PARA_INTERNAL_DPV1.Request_STATUS,
               ENO => #_w2);
   #Request_Sent_32bit := #_w2;
END_REGION

REGION Network 82: Wrtie parameter area DP-V1 for 16-bit parameter type
   RUNG wire#powerrail
      Contact( #PARA_INTERNAL_DPV0.Write_Request )
      Contact( #Drive_Type_Dummy )
      Contact( #Format_Check )
      I_Contact( #Request_Sent_32bit )
      { S7_Templates := "[ptr_type := Variant, id_type := HW_IO, index_type := DInt, len_type := UInt]" } #DPV1_WRITE.WRREC(REQ := wire#w1, ID := #ADR_OUT, INDEX := 47, LEN := 14, RECORD := #PARA_INTERNAL_DPV1_16bit.Request, DONE => #PARA_INTERNAL_DPV1_16bit.Request_DONE, BUSY => #PARA_INTERNAL_DPV1_16bit.Request_BUSY, ERROR => #PARA_INTERNAL_DPV1_16bit.Request_ERROR, STATUS => #PARA_INTERNAL_DPV1_16bit.Request_STATUS)
      Coil( #Request_Sent_16bit_1 )
   END_RUNG
   RUNG wire#powerrail
      Contact( #PARA_INTERNAL_DPV0.Write_Request )
      Contact( #DPV_MODE )
   END_RUNG wire#w1
   // the same network as SCL:
   #_w1 := #PARA_INTERNAL_DPV0.Write_Request AND #Drive_Type_Dummy AND #Format_Check AND NOT #Request_Sent_32bit;
   #DPV1_WRITE(EN := #_w1,   // WRREC
               REQ := #PARA_INTERNAL_DPV0.Write_Request AND #DPV_MODE,
               ID := #ADR_OUT,
               INDEX := 47,
               LEN := 14,
               RECORD := #PARA_INTERNAL_DPV1_16bit.Request,
               DONE => #PARA_INTERNAL_DPV1_16bit.Request_DONE,
               BUSY => #PARA_INTERNAL_DPV1_16bit.Request_BUSY,
               ERROR => #PARA_INTERNAL_DPV1_16bit.Request_ERROR,
               STATUS => #PARA_INTERNAL_DPV1_16bit.Request_STATUS,
               ENO => #_w2);
   #Request_Sent_16bit_1 := #_w2;
END_REGION

REGION Network 83: Responce parameter area DP-V1
   RUNG wire#powerrail
      Contact( #DPV_MODE )
      { S7_Templates := "[ptr_type := Variant, id_type := HW_IO, index_type := DInt, len_type := UInt]" } #DP1_RESPONCE.RDREC(REQ := wire#w1, ID := #ADR_IN, INDEX := 47, MLEN := 10, RECORD := #PARA_INTERNAL_DPV1.Responce, VALID => #PARA_INTERNAL_DPV1.Responce_VALID, BUSY => #PARA_INTERNAL_DPV1.Responce_BUSY, ERROR => #PARA_INTERNAL_DPV1.Responce_ERROR, STATUS => #PARA_INTERNAL_DPV1.Responce_STATUS, LEN => #PARA_INTERNAL_DPV1.Responce_LEN)
   END_RUNG
   RUNG wire#powerrail
      Contact( #DPV_MODE )
      Contact( #PARA_INTERNAL_DPV0.Busy )
      P_Trig( #PARA_INTERNAL_DPV0.Para_27 )
      S_SR(operand := #PARA_INTERNAL_DPV0.Para_28, r1 := #PARA_INTERNAL_DPV1.Responce_VALID)
   END_RUNG wire#w1
   // the same network as SCL:
   #_w1 := #DPV_MODE AND #PARA_INTERNAL_DPV0.Busy;
   #_w2 := #_w1 AND NOT #PARA_INTERNAL_DPV0.Para_27;   // rising edge
   #PARA_INTERNAL_DPV0.Para_27 := #_w1;
   IF #_w2 THEN
       #PARA_INTERNAL_DPV0.Para_28 := TRUE;   // SR flip-flop
   END_IF;
   IF #PARA_INTERNAL_DPV1.Responce_VALID THEN #PARA_INTERNAL_DPV0.Para_28 := FALSE; END_IF;
   IF #DPV_MODE THEN
       #DP1_RESPONCE(REQ := #PARA_INTERNAL_DPV0.Para_28,   // RDREC
                     ID := #ADR_IN,
                     INDEX := 47,
                     MLEN := 10,
                     RECORD := #PARA_INTERNAL_DPV1.Responce,
                     VALID => #PARA_INTERNAL_DPV1.Responce_VALID,
                     BUSY => #PARA_INTERNAL_DPV1.Responce_BUSY,
                     ERROR => #PARA_INTERNAL_DPV1.Responce_ERROR,
                     STATUS => #PARA_INTERNAL_DPV1.Responce_STATUS,
                     LEN => #PARA_INTERNAL_DPV1.Responce_LEN);
   END_IF;
END_REGION
END_FUNCTION_BLOCK

ORGANIZATION_BLOCK "IO"   // OB123, FBD, ProgramCycle
TITLE = "Main Program Sweep (Cycle)"
{ S7_Optimized_Access := 'TRUE' }
// stored: SetENOAutomatically false
   VAR_INPUT
      Initial_Call : Bool;   // Initial call of this OB
      Remanence : Bool;   // =True, if remanent data are available
   END_VAR
   VAR_TEMP
      "101CV1_Temp" : Real;
      "101CV2_Temp" : Real;
   END_VAR
   VAR_TEMP   // added for the SCL form of the ladder/FBD networks
      _w1 : Bool;
   END_VAR
BEGIN

REGION Network 1
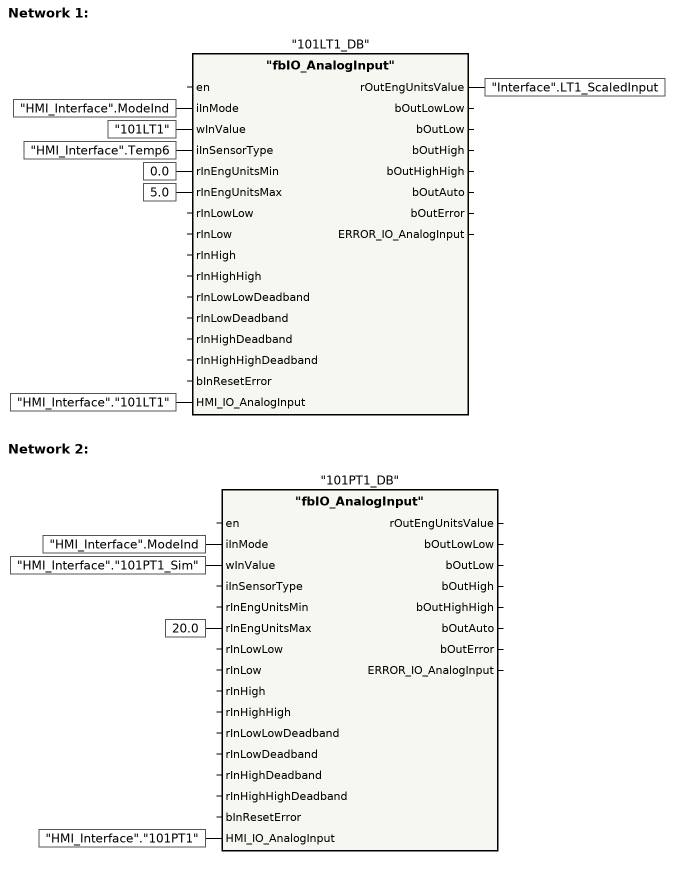
   "101LT1_DB"(iInMode := "HMI_Interface".ModeInd,   // "fbIO_AnalogInput"
               wInValue := "101LT1",
               iInSensorType := "HMI_Interface".Temp6,
               rInEngUnitsMin := 0.0,
               rInEngUnitsMax := 5.0,
               HMI_IO_AnalogInput := "HMI_Interface"."101LT1",
               rOutEngUnitsValue => "Interface".LT1_ScaledInput);
END_REGION

REGION Network 2
   "101PT1_DB"(iInMode := "HMI_Interface".ModeInd,   // "fbIO_AnalogInput"
               wInValue := "HMI_Interface"."101PT1_Sim",
               rInEngUnitsMax := 20.0,
               HMI_IO_AnalogInput := "HMI_Interface"."101PT1");
END_REGION

REGION Network 3: "101CV1
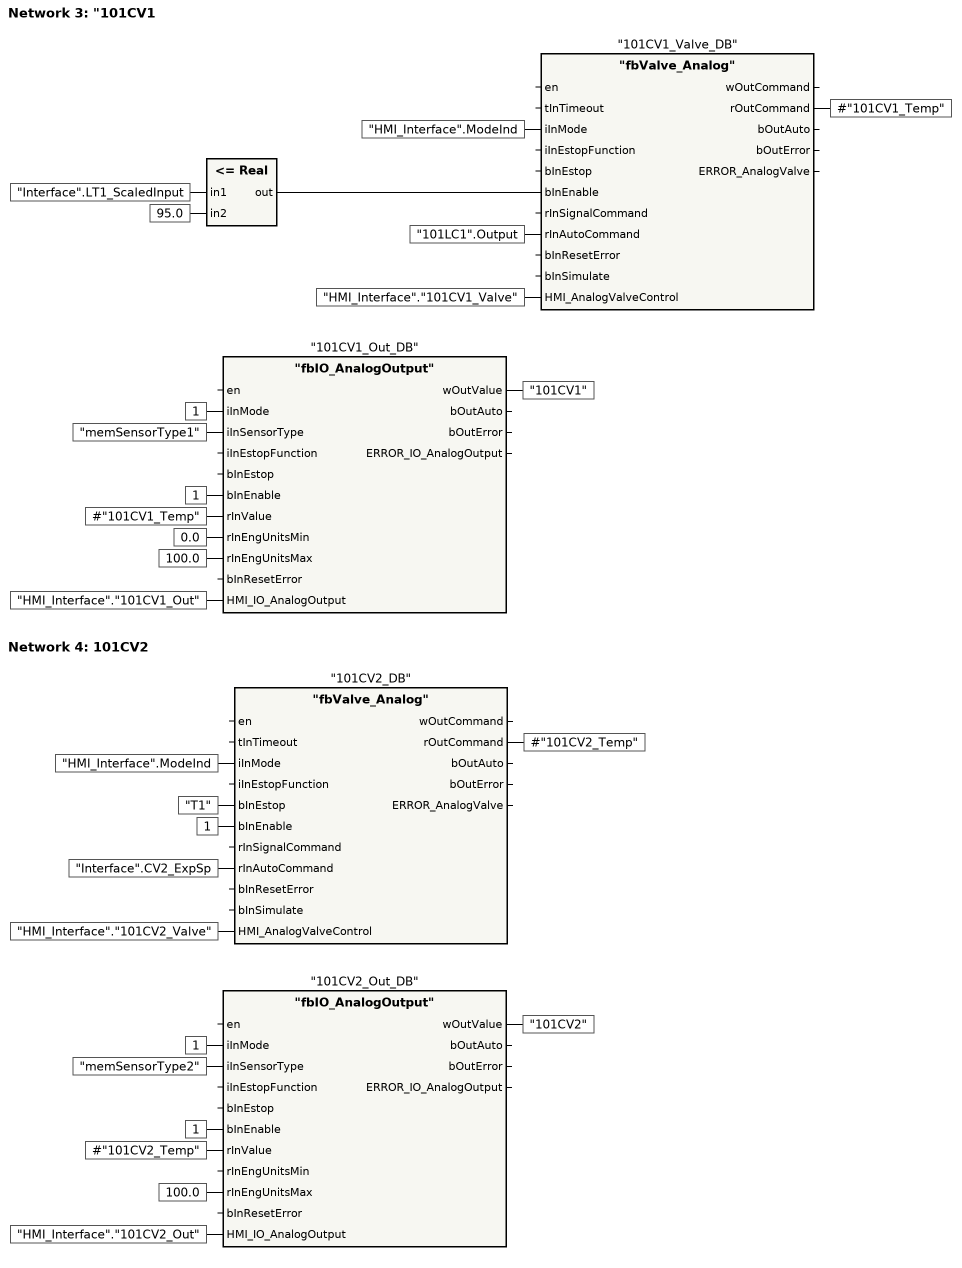
   "101CV1_Valve_DB"(iInMode := "HMI_Interface".ModeInd,   // "fbValve_Analog"
                     bInEnable := "Interface".LT1_ScaledInput <= 95.0,
                     rInAutoCommand := "101LC1".Output,
                     HMI_AnalogValveControl := "HMI_Interface"."101CV1_Valve",
                     rOutCommand => #"101CV1_Temp");
   "101CV1_Out_DB"(iInMode := 1,   // "fbIO_AnalogOutput"
                   iInSensorType := "memSensorType1",
                   bInEnable := 1,
                   rInValue := #"101CV1_Temp",
                   rInEngUnitsMin := 0.0,
                   rInEngUnitsMax := 100.0,
                   HMI_IO_AnalogOutput := "HMI_Interface"."101CV1_Out",
                   wOutValue => "101CV1");
END_REGION

REGION Network 4: 101CV2
   "101CV2_DB"(iInMode := "HMI_Interface".ModeInd,   // "fbValve_Analog"
               bInEstop := "T1",
               bInEnable := 1,
               rInAutoCommand := "Interface".CV2_ExpSp,
               HMI_AnalogValveControl := "HMI_Interface"."101CV2_Valve",
               rOutCommand => #"101CV2_Temp");
   "101CV2_Out_DB"(iInMode := 1,   // "fbIO_AnalogOutput"
                   iInSensorType := "memSensorType2",
                   bInEnable := 1,
                   rInValue := #"101CV2_Temp",
                   rInEngUnitsMax := 100.0,
                   HMI_IO_AnalogOutput := "HMI_Interface"."101CV2_Out",
                   wOutValue => "101CV2");
END_REGION

REGION Network 5: 101DV1
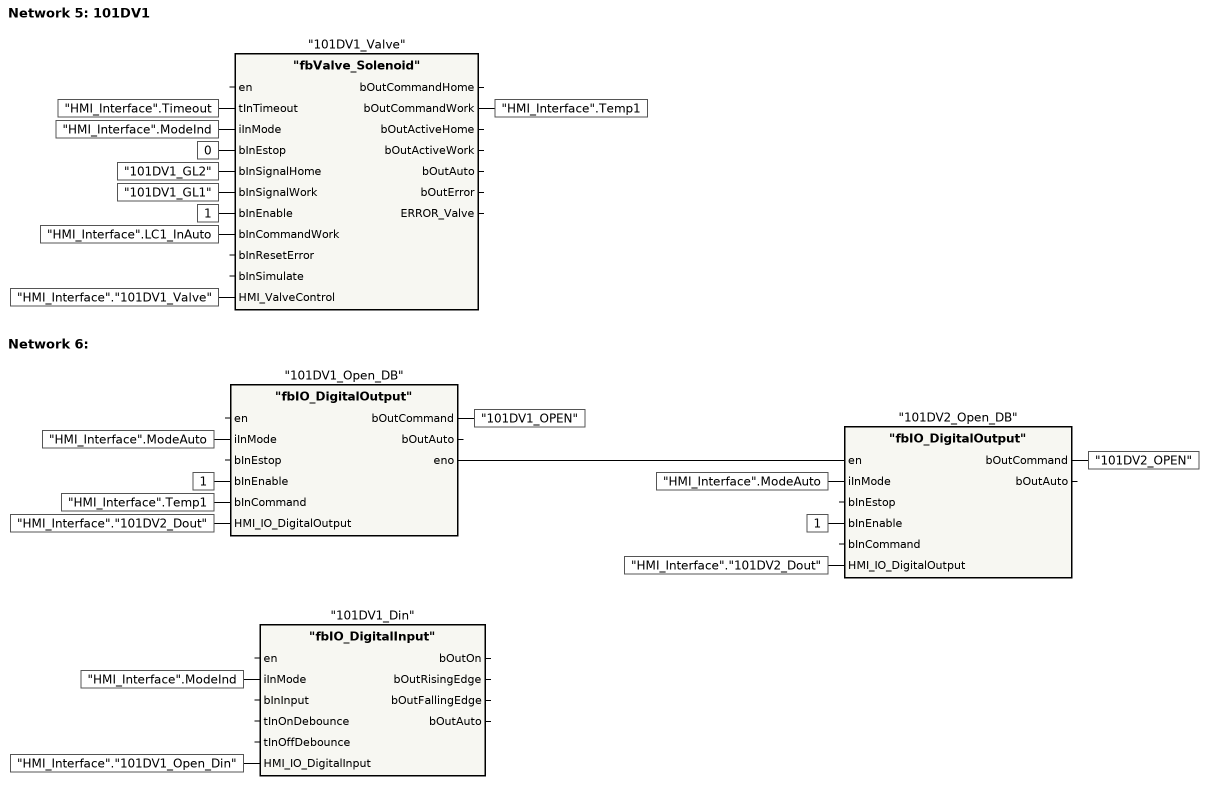
   "101DV1_Valve"(tInTimeout := "HMI_Interface".Timeout,   // "fbValve_Solenoid"
                  iInMode := "HMI_Interface".ModeInd,
                  bInEstop := 0,
                  bInSignalHome := "101DV1_GL2",
                  bInSignalWork := "101DV1_GL1",
                  bInEnable := 1,
                  bInCommandWork := "HMI_Interface".LC1_InAuto,
                  HMI_ValveControl := "HMI_Interface"."101DV1_Valve",
                  bOutCommandWork => "HMI_Interface".Temp1);
END_REGION

REGION Network 6
   "101DV1_Open_DB"(iInMode := "HMI_Interface".ModeAuto,   // "fbIO_DigitalOutput"
                    bInEnable := 1,
                    bInCommand := "HMI_Interface".Temp1,
                    HMI_IO_DigitalOutput := "HMI_Interface"."101DV2_Dout",
                    bOutCommand => "101DV1_OPEN",
                    ENO => #_w1);
   IF #_w1 THEN
       "101DV2_Open_DB"(iInMode := "HMI_Interface".ModeAuto,   // "fbIO_DigitalOutput"
                        bInEnable := 1,
                        HMI_IO_DigitalOutput := "HMI_Interface"."101DV2_Dout",
                        bOutCommand => "101DV2_OPEN");
   END_IF;
   "101DV1_Din"(iInMode := "HMI_Interface".ModeInd, HMI_IO_DigitalInput := "HMI_Interface"."101DV1_Open_Din");   // "fbIO_DigitalInput"
END_REGION
END_ORGANIZATION_BLOCK

ORGANIZATION_BLOCK "PID_Control"   // OB30, FBD, CyclicInterrupt
{ S7_Optimized_Access := 'TRUE' }
// stored: SetENOAutomatically false
   VAR_INPUT
      Initial_Call : Bool;   // Initial call of this OB
      Event_Count : Int;   // Events discarded
   END_VAR
BEGIN

REGION Network 1
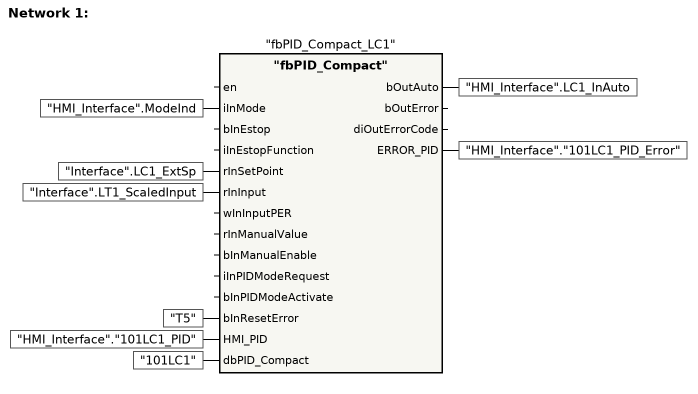
   "fbPID_Compact_LC1"(iInMode := "HMI_Interface".ModeInd,   // "fbPID_Compact"
                       rInSetPoint := "Interface".LC1_ExtSp,
                       rInInput := "Interface".LT1_ScaledInput,
                       bInResetError := "T5",
                       HMI_PID := "HMI_Interface"."101LC1_PID",
                       dbPID_Compact := "101LC1",
                       bOutAuto => "HMI_Interface".LC1_InAuto,
                       ERROR_PID => "HMI_Interface"."101LC1_PID_Error");
END_REGION
END_ORGANIZATION_BLOCK

ORGANIZATION_BLOCK "Sim"   // OB124, FBD, ProgramCycle
TITLE = "Main Program Sweep (Cycle)"
{ S7_Optimized_Access := 'TRUE' }
// stored: SetENOAutomatically false
   VAR_INPUT
      Initial_Call : Bool;   // Initial call of this OB
      Remanence : Bool;   // =True, if remanent data are available
   END_VAR
BEGIN

REGION Network 1
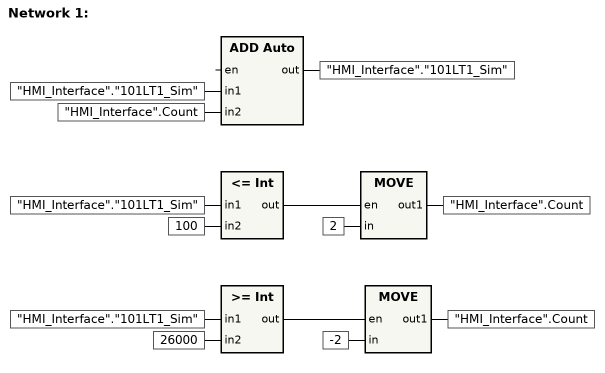
   "HMI_Interface"."101LT1_Sim" := "HMI_Interface"."101LT1_Sim" + "HMI_Interface".Count;
   IF "HMI_Interface"."101LT1_Sim" <= 100 THEN "HMI_Interface".Count := 2; END_IF;
   IF "HMI_Interface"."101LT1_Sim" >= 26000 THEN "HMI_Interface".Count := -2; END_IF;
END_REGION
END_ORGANIZATION_BLOCK

ORGANIZATION_BLOCK "Startup"   // OB100, FBD, Startup
TITLE = "Complete Restart"
{ S7_Optimized_Access := 'TRUE' }
// stored: SetENOAutomatically false
   VAR_INPUT
      LostRetentive : Bool;   // True if retentive data are lost
      LostRTC : Bool;   // True if date and time are lost
   END_VAR
BEGIN

REGION Network 1: Set point for automatic mode LC1 och CV1
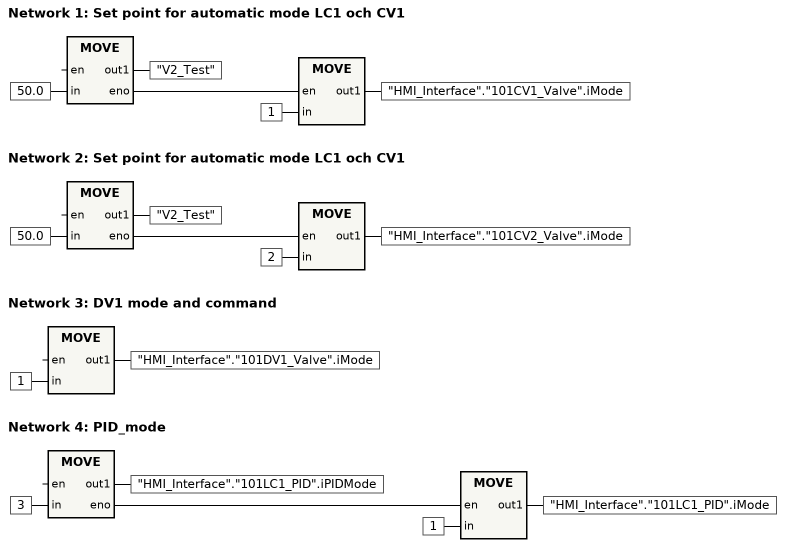
   "V2_Test" := 50.0;
   "HMI_Interface"."101CV1_Valve".iMode := 1;
END_REGION

REGION Network 2: Set point for automatic mode LC1 och CV1
   "V2_Test" := 50.0;
   "HMI_Interface"."101CV2_Valve".iMode := 2;
END_REGION

REGION Network 3: DV1 mode and command
   "HMI_Interface"."101DV1_Valve".iMode := 1;
END_REGION

REGION Network 4: PID_mode
   "HMI_Interface"."101LC1_PID".iPIDMode := 3;
   "HMI_Interface"."101LC1_PID".iMode := 1;
END_REGION
END_ORGANIZATION_BLOCK

ORGANIZATION_BLOCK "Tankcontrol"   // OB125, FBD, ProgramCycle
TITLE = "Main Program Sweep (Cycle)"
{ S7_Optimized_Access := 'TRUE' }
// stored: SetENOAutomatically false
   VAR_INPUT
      Initial_Call : Bool;   // Initial call of this OB
      Remanence : Bool;   // =True, if remanent data are available
   END_VAR
BEGIN
END_ORGANIZATION_BLOCK

FUNCTION "Mapping" : Void
{ S7_Optimized_Access := 'TRUE' }
VERSION : 0.1
   VAR_TEMP 
      Fram : Int;
      Bak : Int;
   END_VAR


BEGIN
	"RH_OUT_2510TR_DB".Control.Fwd_request := "Forward";
	"RH_OUT_2510TR_DB".Control.Rev_request := "Backward";
	"RH_OUT_2510TR_DB"."Status.Ack" := "Acknowledge";
	
	"Status" := "RH_OUT_2510TR_DB".Drive.Status;
	"Alarm" := "RH_OUT_2510TR_DB".Drive.Alarm;
	"Alarm_number" := "RH_OUT_2510TR_DB".Drive.Alarm_number;
	
	//"Forward" := "Fram";
	//"Backward" := "Bak";
	// Här var det skillnad
END_FUNCTION
